PROGRAM MAIN
VAR
	
END_VAR

END_PROGRAM

(* stored: Version 1.1.0.1, ProductVersion 3.1.4024.4
   POU MAIN: Id {536ebec5-64ea-44f4-a7d3-77b57f6c07a7}, SpecialFunc None *)
